FUNCTION_BLOCK fbSensorNoise
VAR_INPUT
	noise_enable:BOOL;
	Ampl        :LREAL;
END_VAR
VAR_OUTPUT
noise_level : LREAL:=0;	
END_VAR
VAR
	fBNoise:FB_CTRL_NOISE_GENERATOR;
	fbNoiseParams: ST_CTRL_NOISE_GENERATOR_PARAMS;
END_VAR

// Generate noise for Sensors ( simulation ) 
fbNoiseParams.tCtrlCycleTime := T#10MS ;
fbNoiseParams.tTaskCycleTime := T#10MS ;
fbNoiseParams.fAmplitude := Ampl;

//
noise_level:=0;
IF Noise_enable THEN
	fbNoise ( fManSyncValue := 1 , eMode := 2 , stParams := fbNoiseParams ) ;
END_IF
noise_level:=fbNoise.fOut;

END_FUNCTION_BLOCK

(* stored: Version 1.1.0.1, ProductVersion 3.1.4024.2
   POU fbSensorNoise: Id {fd77ca23-cff8-4766-99e1-8e930c6d0f01}, SpecialFunc None *)
